INTERFACE IService

END_INTERFACE

(* stored: Version 1.1.0.1
   Itf IService: Id {dd0f70e9-3852-4486-a7e7-cd9998eda431} *)
